# EPICS autosave request: urRobotApp/Db/robotiq_gripper_settings.req
$(P)RobotiqGripper:Units.VAL
$(P)RobotiqGripper:SetPosition.VAL
$(P)RobotiqGripper:SetSpeed.VAL
$(P)RobotiqGripper:SetForce.VAL
